// TIA Portal V20 export
DATA_BLOCK "IdentRfHmi"   // DB213
// stored: MemoryReserve 100
   VAR
      unitIdentRf : Array[0.."NO_OF_UNITS"] of "typeEMIdentRf";
   END_VAR
BEGIN
   unitIdentRf[0].identRfEM[0..7].selectedUnit := 0;
   unitIdentRf[0].identRfEM[0..7].selectedEM := 0;
   unitIdentRf[0].identRfEM[0..7].rfReaderId := 0;
   unitIdentRf[0].identRfEM[0..7].numberOfRf := 0;
   unitIdentRf[0].identRfEM[0].rfReader[0..1].deviceName := WSTRING#'';
   unitIdentRf[0].identRfEM[1].rfReader[0..1].deviceName := WSTRING#'';
   unitIdentRf[0].identRfEM[2].rfReader[0..1].deviceName := WSTRING#'';
   unitIdentRf[0].identRfEM[3].rfReader[0..1].deviceName := WSTRING#'';
   unitIdentRf[0].identRfEM[4].rfReader[0..1].deviceName := WSTRING#'';
   unitIdentRf[0].identRfEM[5].rfReader[0..1].deviceName := WSTRING#'';
   unitIdentRf[0].identRfEM[6].rfReader[0..1].deviceName := WSTRING#'';
   unitIdentRf[0].identRfEM[7].rfReader[0..1].deviceName := WSTRING#'';
   unitIdentRf[0].identRfEM[0].rfReader[0..1].deviceType := WSTRING#'';
   unitIdentRf[0].identRfEM[1].rfReader[0..1].deviceType := WSTRING#'';
   unitIdentRf[0].identRfEM[2].rfReader[0..1].deviceType := WSTRING#'';
   unitIdentRf[0].identRfEM[3].rfReader[0..1].deviceType := WSTRING#'';
   unitIdentRf[0].identRfEM[4].rfReader[0..1].deviceType := WSTRING#'';
   unitIdentRf[0].identRfEM[5].rfReader[0..1].deviceType := WSTRING#'';
   unitIdentRf[0].identRfEM[6].rfReader[0..1].deviceType := WSTRING#'';
   unitIdentRf[0].identRfEM[7].rfReader[0..1].deviceType := WSTRING#'';
   unitIdentRf[0].identRfEM[0].rfReader[0..1].deviceId := 0;
   unitIdentRf[0].identRfEM[1].rfReader[0..1].deviceId := 0;
   unitIdentRf[0].identRfEM[2].rfReader[0..1].deviceId := 0;
   unitIdentRf[0].identRfEM[3].rfReader[0..1].deviceId := 0;
   unitIdentRf[0].identRfEM[4].rfReader[0..1].deviceId := 0;
   unitIdentRf[0].identRfEM[5].rfReader[0..1].deviceId := 0;
   unitIdentRf[0].identRfEM[6].rfReader[0..1].deviceId := 0;
   unitIdentRf[0].identRfEM[7].rfReader[0..1].deviceId := 0;
   unitIdentRf[0].identRfEM[0].rfReader[0..1].tagType := WSTRING#'';
   unitIdentRf[0].identRfEM[1].rfReader[0..1].tagType := WSTRING#'';
   unitIdentRf[0].identRfEM[2].rfReader[0..1].tagType := WSTRING#'';
   unitIdentRf[0].identRfEM[3].rfReader[0..1].tagType := WSTRING#'';
   unitIdentRf[0].identRfEM[4].rfReader[0..1].tagType := WSTRING#'';
   unitIdentRf[0].identRfEM[5].rfReader[0..1].tagType := WSTRING#'';
   unitIdentRf[0].identRfEM[6].rfReader[0..1].tagType := WSTRING#'';
   unitIdentRf[0].identRfEM[7].rfReader[0..1].tagType := WSTRING#'';
   unitIdentRf[0].identRfEM[0].rfReader[0..1].cameraMode := WSTRING#'';
   unitIdentRf[0].identRfEM[1].rfReader[0..1].cameraMode := WSTRING#'';
   unitIdentRf[0].identRfEM[2].rfReader[0..1].cameraMode := WSTRING#'';
   unitIdentRf[0].identRfEM[3].rfReader[0..1].cameraMode := WSTRING#'';
   unitIdentRf[0].identRfEM[4].rfReader[0..1].cameraMode := WSTRING#'';
   unitIdentRf[0].identRfEM[5].rfReader[0..1].cameraMode := WSTRING#'';
   unitIdentRf[0].identRfEM[6].rfReader[0..1].cameraMode := WSTRING#'';
   unitIdentRf[0].identRfEM[7].rfReader[0..1].cameraMode := WSTRING#'';
   unitIdentRf[0].identRfEM[0].rfReader[0..1].resultState := WSTRING#'';
   unitIdentRf[0].identRfEM[1].rfReader[0..1].resultState := WSTRING#'';
   unitIdentRf[0].identRfEM[2].rfReader[0..1].resultState := WSTRING#'';
   unitIdentRf[0].identRfEM[3].rfReader[0..1].resultState := WSTRING#'';
   unitIdentRf[0].identRfEM[4].rfReader[0..1].resultState := WSTRING#'';
   unitIdentRf[0].identRfEM[5].rfReader[0..1].resultState := WSTRING#'';
   unitIdentRf[0].identRfEM[6].rfReader[0..1].resultState := WSTRING#'';
   unitIdentRf[0].identRfEM[7].rfReader[0..1].resultState := WSTRING#'';
   unitIdentRf[0].identRfEM[0].rfReader[0..1].progNo := 0;
   unitIdentRf[0].identRfEM[1].rfReader[0..1].progNo := 0;
   unitIdentRf[0].identRfEM[2].rfReader[0..1].progNo := 0;
   unitIdentRf[0].identRfEM[3].rfReader[0..1].progNo := 0;
   unitIdentRf[0].identRfEM[4].rfReader[0..1].progNo := 0;
   unitIdentRf[0].identRfEM[5].rfReader[0..1].progNo := 0;
   unitIdentRf[0].identRfEM[6].rfReader[0..1].progNo := 0;
   unitIdentRf[0].identRfEM[7].rfReader[0..1].progNo := 0;
   unitIdentRf[0].identRfEM[0].rfReader[0..1].progNumberWrite := 0;
   unitIdentRf[0].identRfEM[1].rfReader[0..1].progNumberWrite := 0;
   unitIdentRf[0].identRfEM[2].rfReader[0..1].progNumberWrite := 0;
   unitIdentRf[0].identRfEM[3].rfReader[0..1].progNumberWrite := 0;
   unitIdentRf[0].identRfEM[4].rfReader[0..1].progNumberWrite := 0;
   unitIdentRf[0].identRfEM[5].rfReader[0..1].progNumberWrite := 0;
   unitIdentRf[0].identRfEM[6].rfReader[0..1].progNumberWrite := 0;
   unitIdentRf[0].identRfEM[7].rfReader[0..1].progNumberWrite := 0;
   unitIdentRf[0].identRfEM[0].rfReader[0..1].pushbutton := 16#0000;
   unitIdentRf[0].identRfEM[1].rfReader[0..1].pushbutton := 16#0000;
   unitIdentRf[0].identRfEM[2].rfReader[0..1].pushbutton := 16#0000;
   unitIdentRf[0].identRfEM[3].rfReader[0..1].pushbutton := 16#0000;
   unitIdentRf[0].identRfEM[4].rfReader[0..1].pushbutton := 16#0000;
   unitIdentRf[0].identRfEM[5].rfReader[0..1].pushbutton := 16#0000;
   unitIdentRf[0].identRfEM[6].rfReader[0..1].pushbutton := 16#0000;
   unitIdentRf[0].identRfEM[7].rfReader[0..1].pushbutton := 16#0000;
   unitIdentRf[0].identRfEM[0].rfReader[0..1].enablePushbutton := 16#0000;
   unitIdentRf[0].identRfEM[1].rfReader[0..1].enablePushbutton := 16#0000;
   unitIdentRf[0].identRfEM[2].rfReader[0..1].enablePushbutton := 16#0000;
   unitIdentRf[0].identRfEM[3].rfReader[0..1].enablePushbutton := 16#0000;
   unitIdentRf[0].identRfEM[4].rfReader[0..1].enablePushbutton := 16#0000;
   unitIdentRf[0].identRfEM[5].rfReader[0..1].enablePushbutton := 16#0000;
   unitIdentRf[0].identRfEM[6].rfReader[0..1].enablePushbutton := 16#0000;
   unitIdentRf[0].identRfEM[7].rfReader[0..1].enablePushbutton := 16#0000;
   unitIdentRf[0].identRfEM[0].rfReader[0..1].status := 16#0000;
   unitIdentRf[0].identRfEM[1].rfReader[0..1].status := 16#0000;
   unitIdentRf[0].identRfEM[2].rfReader[0..1].status := 16#0000;
   unitIdentRf[0].identRfEM[3].rfReader[0..1].status := 16#0000;
   unitIdentRf[0].identRfEM[4].rfReader[0..1].status := 16#0000;
   unitIdentRf[0].identRfEM[5].rfReader[0..1].status := 16#0000;
   unitIdentRf[0].identRfEM[6].rfReader[0..1].status := 16#0000;
   unitIdentRf[0].identRfEM[7].rfReader[0..1].status := 16#0000;
   unitIdentRf[0].identRfEM[0].rfReader[0..1].alarmCategorie := 0;
   unitIdentRf[0].identRfEM[1].rfReader[0..1].alarmCategorie := 0;
   unitIdentRf[0].identRfEM[2].rfReader[0..1].alarmCategorie := 0;
   unitIdentRf[0].identRfEM[3].rfReader[0..1].alarmCategorie := 0;
   unitIdentRf[0].identRfEM[4].rfReader[0..1].alarmCategorie := 0;
   unitIdentRf[0].identRfEM[5].rfReader[0..1].alarmCategorie := 0;
   unitIdentRf[0].identRfEM[6].rfReader[0..1].alarmCategorie := 0;
   unitIdentRf[0].identRfEM[7].rfReader[0..1].alarmCategorie := 0;
   unitIdentRf[0].identRfEM[0].rfReader[0..1].alarmNo := 0;
   unitIdentRf[0].identRfEM[1].rfReader[0..1].alarmNo := 0;
   unitIdentRf[0].identRfEM[2].rfReader[0..1].alarmNo := 0;
   unitIdentRf[0].identRfEM[3].rfReader[0..1].alarmNo := 0;
   unitIdentRf[0].identRfEM[4].rfReader[0..1].alarmNo := 0;
   unitIdentRf[0].identRfEM[5].rfReader[0..1].alarmNo := 0;
   unitIdentRf[0].identRfEM[6].rfReader[0..1].alarmNo := 0;
   unitIdentRf[0].identRfEM[7].rfReader[0..1].alarmNo := 0;
   unitIdentRf[0].identRfEM[0].rfReader[0..1].alarmCode := 16#0000_0000;
   unitIdentRf[0].identRfEM[1].rfReader[0..1].alarmCode := 16#0000_0000;
   unitIdentRf[0].identRfEM[2].rfReader[0..1].alarmCode := 16#0000_0000;
   unitIdentRf[0].identRfEM[3].rfReader[0..1].alarmCode := 16#0000_0000;
   unitIdentRf[0].identRfEM[4].rfReader[0..1].alarmCode := 16#0000_0000;
   unitIdentRf[0].identRfEM[5].rfReader[0..1].alarmCode := 16#0000_0000;
   unitIdentRf[0].identRfEM[6].rfReader[0..1].alarmCode := 16#0000_0000;
   unitIdentRf[0].identRfEM[7].rfReader[0..1].alarmCode := 16#0000_0000;
   unitIdentRf[0].identRfEM[0].rfReader[0..1].resultColor := 0;
   unitIdentRf[0].identRfEM[1].rfReader[0..1].resultColor := 0;
   unitIdentRf[0].identRfEM[2].rfReader[0..1].resultColor := 0;
   unitIdentRf[0].identRfEM[3].rfReader[0..1].resultColor := 0;
   unitIdentRf[0].identRfEM[4].rfReader[0..1].resultColor := 0;
   unitIdentRf[0].identRfEM[5].rfReader[0..1].resultColor := 0;
   unitIdentRf[0].identRfEM[6].rfReader[0..1].resultColor := 0;
   unitIdentRf[0].identRfEM[7].rfReader[0..1].resultColor := 0;
   unitIdentRf[0].identRfEM[0].rfReader[0..1].statusColorCode := 0;
   unitIdentRf[0].identRfEM[1].rfReader[0..1].statusColorCode := 0;
   unitIdentRf[0].identRfEM[2].rfReader[0..1].statusColorCode := 0;
   unitIdentRf[0].identRfEM[3].rfReader[0..1].statusColorCode := 0;
   unitIdentRf[0].identRfEM[4].rfReader[0..1].statusColorCode := 0;
   unitIdentRf[0].identRfEM[5].rfReader[0..1].statusColorCode := 0;
   unitIdentRf[0].identRfEM[6].rfReader[0..1].statusColorCode := 0;
   unitIdentRf[0].identRfEM[7].rfReader[0..1].statusColorCode := 0;
   unitIdentRf[0].identRfEM[0].rfReader[0..1].datRead1 := '';
   unitIdentRf[0].identRfEM[1].rfReader[0..1].datRead1 := '';
   unitIdentRf[0].identRfEM[2].rfReader[0..1].datRead1 := '';
   unitIdentRf[0].identRfEM[3].rfReader[0..1].datRead1 := '';
   unitIdentRf[0].identRfEM[4].rfReader[0..1].datRead1 := '';
   unitIdentRf[0].identRfEM[5].rfReader[0..1].datRead1 := '';
   unitIdentRf[0].identRfEM[6].rfReader[0..1].datRead1 := '';
   unitIdentRf[0].identRfEM[7].rfReader[0..1].datRead1 := '';
   unitIdentRf[0].identRfEM[0].rfReader[0..1].datRead2 := '';
   unitIdentRf[0].identRfEM[1].rfReader[0..1].datRead2 := '';
   unitIdentRf[0].identRfEM[2].rfReader[0..1].datRead2 := '';
   unitIdentRf[0].identRfEM[3].rfReader[0..1].datRead2 := '';
   unitIdentRf[0].identRfEM[4].rfReader[0..1].datRead2 := '';
   unitIdentRf[0].identRfEM[5].rfReader[0..1].datRead2 := '';
   unitIdentRf[0].identRfEM[6].rfReader[0..1].datRead2 := '';
   unitIdentRf[0].identRfEM[7].rfReader[0..1].datRead2 := '';
   unitIdentRf[0].identRfEM[0].rfReader[0..1].datRead3 := '';
   unitIdentRf[0].identRfEM[1].rfReader[0..1].datRead3 := '';
   unitIdentRf[0].identRfEM[2].rfReader[0..1].datRead3 := '';
   unitIdentRf[0].identRfEM[3].rfReader[0..1].datRead3 := '';
   unitIdentRf[0].identRfEM[4].rfReader[0..1].datRead3 := '';
   unitIdentRf[0].identRfEM[5].rfReader[0..1].datRead3 := '';
   unitIdentRf[0].identRfEM[6].rfReader[0..1].datRead3 := '';
   unitIdentRf[0].identRfEM[7].rfReader[0..1].datRead3 := '';
   unitIdentRf[0].identRfEM[0].rfReader[0..1].datRead4 := '';
   unitIdentRf[0].identRfEM[1].rfReader[0..1].datRead4 := '';
   unitIdentRf[0].identRfEM[2].rfReader[0..1].datRead4 := '';
   unitIdentRf[0].identRfEM[3].rfReader[0..1].datRead4 := '';
   unitIdentRf[0].identRfEM[4].rfReader[0..1].datRead4 := '';
   unitIdentRf[0].identRfEM[5].rfReader[0..1].datRead4 := '';
   unitIdentRf[0].identRfEM[6].rfReader[0..1].datRead4 := '';
   unitIdentRf[0].identRfEM[7].rfReader[0..1].datRead4 := '';
   unitIdentRf[0].identRfEM[0].rfReader[0..1].datWrite1 := '';
   unitIdentRf[0].identRfEM[1].rfReader[0..1].datWrite1 := '';
   unitIdentRf[0].identRfEM[2].rfReader[0..1].datWrite1 := '';
   unitIdentRf[0].identRfEM[3].rfReader[0..1].datWrite1 := '';
   unitIdentRf[0].identRfEM[4].rfReader[0..1].datWrite1 := '';
   unitIdentRf[0].identRfEM[5].rfReader[0..1].datWrite1 := '';
   unitIdentRf[0].identRfEM[6].rfReader[0..1].datWrite1 := '';
   unitIdentRf[0].identRfEM[7].rfReader[0..1].datWrite1 := '';
   unitIdentRf[0].identRfEM[0].rfReader[0..1].datWrite2 := '';
   unitIdentRf[0].identRfEM[1].rfReader[0..1].datWrite2 := '';
   unitIdentRf[0].identRfEM[2].rfReader[0..1].datWrite2 := '';
   unitIdentRf[0].identRfEM[3].rfReader[0..1].datWrite2 := '';
   unitIdentRf[0].identRfEM[4].rfReader[0..1].datWrite2 := '';
   unitIdentRf[0].identRfEM[5].rfReader[0..1].datWrite2 := '';
   unitIdentRf[0].identRfEM[6].rfReader[0..1].datWrite2 := '';
   unitIdentRf[0].identRfEM[7].rfReader[0..1].datWrite2 := '';
   unitIdentRf[0].identRfEM[0].rfReader[0..1].datWrite3 := '';
   unitIdentRf[0].identRfEM[1].rfReader[0..1].datWrite3 := '';
   unitIdentRf[0].identRfEM[2].rfReader[0..1].datWrite3 := '';
   unitIdentRf[0].identRfEM[3].rfReader[0..1].datWrite3 := '';
   unitIdentRf[0].identRfEM[4].rfReader[0..1].datWrite3 := '';
   unitIdentRf[0].identRfEM[5].rfReader[0..1].datWrite3 := '';
   unitIdentRf[0].identRfEM[6].rfReader[0..1].datWrite3 := '';
   unitIdentRf[0].identRfEM[7].rfReader[0..1].datWrite3 := '';
   unitIdentRf[0].identRfEM[0].rfReader[0..1].datWrite4 := '';
   unitIdentRf[0].identRfEM[1].rfReader[0..1].datWrite4 := '';
   unitIdentRf[0].identRfEM[2].rfReader[0..1].datWrite4 := '';
   unitIdentRf[0].identRfEM[3].rfReader[0..1].datWrite4 := '';
   unitIdentRf[0].identRfEM[4].rfReader[0..1].datWrite4 := '';
   unitIdentRf[0].identRfEM[5].rfReader[0..1].datWrite4 := '';
   unitIdentRf[0].identRfEM[6].rfReader[0..1].datWrite4 := '';
   unitIdentRf[0].identRfEM[7].rfReader[0..1].datWrite4 := '';
END_DATA_BLOCK
